FUNCTION_BLOCK System
VAR_INPUT CONSTANT
	eOrigin : E_Origin;
END_VAR
VAR_OUTPUT
END_VAR
VAR
	fbTime : FB_LocalSystemTime := ( bEnable := TRUE, dwCycle := 1 );
END_VAR

fbTime();

END_FUNCTION_BLOCK

(* stored: Version 1.1.0.1, ProductVersion 3.1.4024.0
   POU System: Id {602cf87f-f724-402c-a908-37c85e996734}, SpecialFunc None *)
